// TIA Portal V19 export
TYPE "TAx_Warnings"
// stored: Access Published
   STRUCT
      TOAxis : Bool;   // Warning in technology object
      Drive : Bool;   // Warning in drive
   END_STRUCT;
END_TYPE
